FUNCTION_BLOCK FB_JamDetect
VAR_INPUT
	In_PE:	BOOL;		// Photo Eye Input
	In_Status:	BOOL;		// Status to determine if Timer should run (like running status or State) (1=Watch for Jams)
	CFG_PEOKState:	BOOL;		// Photo OK State ( State of Photo Eye for OK or Not blocked State State (1 or 0))
	JamDetTime: TIME;		// Time to wait before sending Jam detected Output
END_VAR
VAR_OUTPUT
	JamDetected:	BOOL;		// Out for Jam detected
END_VAR
VAR
	PhotoEyeBlocked: BOOL;
	JamTimer: TON;
	JamWatchEnable: BOOL;
	PE_ClearTrig: F_TRIG;
END_VAR

PhotoEyeBlocked := In_PE XOR CFG_PEOKState;
JamWatchEnable := In_Status AND PhotoEyeBlocked;

JamTimer(IN:= JamWatchEnable, PT:= JamDetTime , Q=>  , ET=> );

IF JamTimer.Q THEN
	JamDetected := TRUE;
END_IF

PE_ClearTrig(CLK:= PhotoEyeBlocked);

IF PE_ClearTrig.Q AND JamDetected THEN
	JamDetected := FALSE;
END_IF

END_FUNCTION_BLOCK

(* stored: Version 1.1.0.1, ProductVersion 3.1.4024.4
   POU FB_JamDetect: Id {25129f8a-700b-45bd-98e0-3a5feef9be4d}, SpecialFunc None *)
